// TIA Portal V20 export
// export: Created 2026-04-10T22:01:57.8237529Z, ExportSetting WithDefaults, DisplayName Totally Integrated Automation Portal, DisplayVersion V20, DisplayName TIA Portal Openness, DisplayVersion V20, DisplayName TIA Portal Version Control Interface, DisplayVersion V20, DisplayName STEP 7 Professional, DisplayVersion V20, DisplayName STEP 7 Safety, DisplayVersion V20, DisplayName WinCC Basic/Comfort/Advanced, DisplayVersion V20
VAR_GLOBAL   // PLC tag table "MOD_"
END_VAR
VAR_GLOBAL CONSTANT   // user constants
   MOD_TP307 : Int := 1;   // Kommentar TP307 / Comment TP307
   MOD_TP308 : Int := 2;   // Kommentar TP308 / Comment TP308
END_VAR
